SUBAPPLICATION MechatronicArm (* Subapplication Type *)
  (* Standard: 61499-2 *)
  (* Version 1.0, 2025-03-21, AK123700 *)
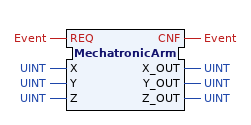
  EVENT_INPUT
    REQ; (* Normal Execution Request *)
  END_EVENT
  EVENT_OUTPUT
    CNF; (* Execution Confirmation *)
  END_EVENT
  VAR_INPUT
    X : UINT;
    Y : UINT;
    Z : UINT;
  END_VAR
  VAR_OUTPUT
    X_OUT : UINT;
    Y_OUT : UINT;
    Z_OUT : UINT;
  END_VAR
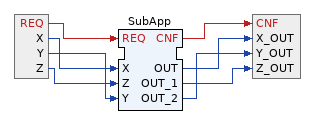
  SUBAPPLICATION SubApp
    EVENT_INPUT
      REQ;
    END_EVENT
    EVENT_OUTPUT
      CNF;
    END_EVENT
    VAR_INPUT
      X : UINT;
      Z : UINT;
      Y : UINT;
    END_VAR
    VAR_OUTPUT
      OUT : UINT;
      OUT_1 : UINT;
      OUT_2 : UINT;
    END_VAR
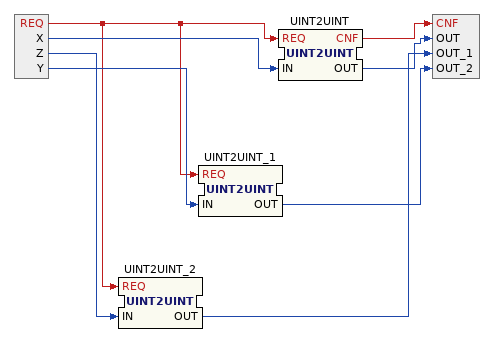
    FBS
      UINT2UINT : UINT2UINT;
      UINT2UINT_2 : UINT2UINT;
      UINT2UINT_1 : UINT2UINT;
    END_FBS
    EVENT_CONNECTIONS
      REQ TO UINT2UINT.REQ;
      UINT2UINT.CNF TO CNF;
      REQ TO UINT2UINT_2.REQ;
      REQ TO UINT2UINT_1.REQ;
    END_CONNECTIONS
    DATA_CONNECTIONS
      X TO UINT2UINT.IN;
      UINT2UINT.OUT TO OUT;
      Z TO UINT2UINT_2.IN;
      UINT2UINT_2.OUT TO OUT_1;
      Y TO UINT2UINT_1.IN;
      UINT2UINT_1.OUT TO OUT_2;
    END_CONNECTIONS
  END_SUBAPPLICATION
  EVENT_CONNECTIONS
    REQ TO SubApp.REQ;
    SubApp.CNF TO CNF;
  END_CONNECTIONS
  DATA_CONNECTIONS
    X TO SubApp.X;
    SubApp.OUT TO X_OUT;
    Z TO SubApp.Z;
    SubApp.OUT_1 TO Z_OUT;
    Y TO SubApp.Y;
    SubApp.OUT_2 TO Y_OUT;
  END_CONNECTIONS
END_SUBAPPLICATION
